{attribute 'qualified_only'}
VAR_GLOBAL
	
	ob_PN_output AT %Q*: BOOL;
	
END_VAR

(* stored: Version 1.1.0.1, ProductVersion 3.1.4024.2
   GVL GVL_PN: Id {4bb8255b-f7b8-40ad-b06e-830a25cddfde} *)
